// TIA Portal V18 export
DATA_BLOCK "_SPOT_DB"   // DB10
{ S7_Optimized_Access := 'TRUE' }
VERSION : 0.1
// stored: AutoNumber true, DBAccessibleFromOPCUA true, IsOnlyStoredInLoadMemory false, IsRetainMemResEnabled false, IsWriteProtectedInAS false, MemoryReserve 100
   VAR
      Spot_i : Int := 0;
      Spot_N_max : Int := 30;
      SpotListNow { S7_SetPoint := 'True'} : "typeSpotList";
   END_VAR
   VAR RETAIN
      Part_selected : Int := 0;
      Part_N : Int;
      Part_N_max : Int := 30;
      Parts { S7_SetPoint := 'True'} : Array[1..10] of "typeSpotList";
   END_VAR
BEGIN
   SpotListNow.N := 4;
   SpotListNow.pos_AR[1].M1Z := 11.0;
   SpotListNow.pos_AR[2].M1Z := 22.0;
   SpotListNow.pos_AR[3].M1Z := 33.0;
   SpotListNow.pos_AR[4..30].M1Z := 0.0;
   SpotListNow.pos_AR[1].M2Y := 11.0;
   SpotListNow.pos_AR[2].M2Y := 22.0;
   SpotListNow.pos_AR[3].M2Y := 33.0;
   SpotListNow.pos_AR[4..30].M2Y := 0.0;
   SpotListNow.pos_AR[1].M3X := 11.0;
   SpotListNow.pos_AR[2].M3X := 22.0;
   SpotListNow.pos_AR[3].M3X := 33.0;
   SpotListNow.pos_AR[4..30].M3X := 0.0;
   SpotListNow.pos_AR[1].M4O1 := 11.0;
   SpotListNow.pos_AR[2].M4O1 := 22.0;
   SpotListNow.pos_AR[3].M4O1 := 33.0;
   SpotListNow.pos_AR[4..30].M4O1 := 0.0;
   SpotListNow.pos_AR[1].M5O2 := 11.0;
   SpotListNow.pos_AR[2].M5O2 := 22.0;
   SpotListNow.pos_AR[3].M5O2 := 33.0;
   SpotListNow.pos_AR[4..30].M5O2 := 0.0;
   Parts[1..10].N := 0;
   Parts[1].pos_AR[1..30].M1Z := 0.0;
   Parts[2].pos_AR[1..30].M1Z := 0.0;
   Parts[3].pos_AR[1..30].M1Z := 0.0;
   Parts[4].pos_AR[1..30].M1Z := 0.0;
   Parts[5].pos_AR[1..30].M1Z := 0.0;
   Parts[6].pos_AR[1..30].M1Z := 0.0;
   Parts[7].pos_AR[1..30].M1Z := 0.0;
   Parts[8].pos_AR[1..30].M1Z := 0.0;
   Parts[9].pos_AR[1..30].M1Z := 0.0;
   Parts[10].pos_AR[1..30].M1Z := 0.0;
   Parts[1].pos_AR[1..30].M2Y := 0.0;
   Parts[2].pos_AR[1..30].M2Y := 0.0;
   Parts[3].pos_AR[1..30].M2Y := 0.0;
   Parts[4].pos_AR[1..30].M2Y := 0.0;
   Parts[5].pos_AR[1..30].M2Y := 0.0;
   Parts[6].pos_AR[1..30].M2Y := 0.0;
   Parts[7].pos_AR[1..30].M2Y := 0.0;
   Parts[8].pos_AR[1..30].M2Y := 0.0;
   Parts[9].pos_AR[1..30].M2Y := 0.0;
   Parts[10].pos_AR[1..30].M2Y := 0.0;
   Parts[1].pos_AR[1..30].M3X := 0.0;
   Parts[2].pos_AR[1..30].M3X := 0.0;
   Parts[3].pos_AR[1..30].M3X := 0.0;
   Parts[4].pos_AR[1..30].M3X := 0.0;
   Parts[5].pos_AR[1..30].M3X := 0.0;
   Parts[6].pos_AR[1..30].M3X := 0.0;
   Parts[7].pos_AR[1..30].M3X := 0.0;
   Parts[8].pos_AR[1..30].M3X := 0.0;
   Parts[9].pos_AR[1..30].M3X := 0.0;
   Parts[10].pos_AR[1..30].M3X := 0.0;
   Parts[1].pos_AR[1..30].M4O1 := 0.0;
   Parts[2].pos_AR[1..30].M4O1 := 0.0;
   Parts[3].pos_AR[1..30].M4O1 := 0.0;
   Parts[4].pos_AR[1..30].M4O1 := 0.0;
   Parts[5].pos_AR[1..30].M4O1 := 0.0;
   Parts[6].pos_AR[1..30].M4O1 := 0.0;
   Parts[7].pos_AR[1..30].M4O1 := 0.0;
   Parts[8].pos_AR[1..30].M4O1 := 0.0;
   Parts[9].pos_AR[1..30].M4O1 := 0.0;
   Parts[10].pos_AR[1..30].M4O1 := 0.0;
   Parts[1].pos_AR[1..30].M5O2 := 0.0;
   Parts[2].pos_AR[1..30].M5O2 := 0.0;
   Parts[3].pos_AR[1..30].M5O2 := 0.0;
   Parts[4].pos_AR[1..30].M5O2 := 0.0;
   Parts[5].pos_AR[1..30].M5O2 := 0.0;
   Parts[6].pos_AR[1..30].M5O2 := 0.0;
   Parts[7].pos_AR[1..30].M5O2 := 0.0;
   Parts[8].pos_AR[1..30].M5O2 := 0.0;
   Parts[9].pos_AR[1..30].M5O2 := 0.0;
   Parts[10].pos_AR[1..30].M5O2 := 0.0;
END_DATA_BLOCK
